{attribute 'qualified_only'}
{attribute 'strict'}
TYPE Resolution :
(
	Invalid := 0,
	_12Bit := 1,
	_16Bit := 2,
	_24Bit := 3
);
END_TYPE

(* stored: Version 1.1.0.1, ProductVersion 3.1.4024.5
   DUT Resolution: Id {8a5e6cee-34c1-4f68-a47b-67841360236e} *)
